// TIA Portal V20 export
FUNCTION_BLOCK "FONCTION"   // FB2, LAD
// stored: MemoryReserve 100, Namespace Ely_2, SetENOAutomatically false
BEGIN
END_FUNCTION_BLOCK
